(* This function use for BurnerControlEcoFlam
| this version dont have Reset components like Digital output, user have to reset manual at the BurnerControlEcoFlam device
*)
FUNCTION_BLOCK FB_BurnerControlEcoFlam IMPLEMENTS I_BurnerControlEcoFlam

VAR
	piFault	: FB_DigitalInput;
	piFireSussess : FB_DigitalInputExt;
	ifActivePower : I_ActivePower;					//have FB
	ifActivePowerNoFB : I_ActivePowerNoFB;
	eActivePowerType : E_ActivePowerType;
	eState	: E_EcoFlamState;
	bAbort: BOOL;
	bBusy: BOOL;
	bInit: BOOL;
	bReset: BOOL;
	bStop: BOOL;
	bError : BOOL;
	tMeasurement	: TIME := T#200S;
	bIgnition: BOOL;
	bIgnitioned: BOOL;
	tonMeasurementTimer: Ton;
	tBurnSuccess: TIME;
	sName : STRING;
END_VAR

bError := piFault.In; //OR piFireSussess.ErrorTimedout;
piFireSussess();
StateMachine();
tonMeasurementTimer(PT := tMeasurement);
IF piFireSussess.RisingTrigger AND eState = ECOFLAM_IGNITION THEN
	tBurnSuccess	:= 	tonMeasurementTimer.ET;				
END_IF

PROPERTY ActivePowerType : Reference to E_ActivePowerType
GET
ActivePowerType ref= eActivePowerType;
END_GET
END_PROPERTY

{attribute 'monitoring' := 'variable'}
PROPERTY Busy : reference to bool
GET
Busy ref= bBusy;
END_GET
END_PROPERTY

PROPERTY Error : REFERENCE to bool
GET
error REF= bError;
END_GET
END_PROPERTY

{attribute 'monitoring' := 'variable'}
PROPERTY IgnitionSucess : bool
GET
CASE eActivePowerType OF
	ACTIVE_POWER_TYPE_NO_FEEDBACK:
		IgnitionSucess := piFireSussess.In AND ifActivePowerNoFB.PowerOnIsCalled;
		
	ACTIVE_POWER_TYPE_FEEDBACK:
		IgnitionSucess := piFireSussess.In AND ifActivePower.PowerOnIsCalled;
END_CASE
END_GET
END_PROPERTY

PROPERTY Inited : bool
GET
Inited := eState=ECOFLAM_READY_INITIALIZED;
END_GET
END_PROPERTY

PROPERTY IsRefActivePower : bool
GET
IsRefActivePower := ifActivePower<>0 OR ifActivePowerNoFB<>0;
END_GET
END_PROPERTY

PROPERTY IsStop : bool
GET
CASE eActivePowerType OF
	ACTIVE_POWER_TYPE_NO_FEEDBACK:
		isStop := ifActivePowerNoFB.PowerOffIsCalled;
		
	ACTIVE_POWER_TYPE_FEEDBACK:
		isStop := NOT ifActivePower.Powered;
END_CASE
END_GET
END_PROPERTY

METHOD MR_Abort : BOOL
VAR_INPUT
END_VAR
IF eState >= ECOFLAM_INITIALIZING THEN
	bAbort := TRUE;
	bBusy := TRUE;
	MR_Abort := FALSE;
	eState := ECOFLAM_ABORTING;
ELSIF eState = ECOFLAM_UNINITIALIZED THEN
	bAbort := FALSE;
	bBusy := FALSE;
	MR_Abort := TRUE;
END_IF
END_METHOD

METHOD MR_AppendPowerOn : BOOL
VAR_INPUT
	iPowerON	: I_ActivePower;
END_VAR
IF THIS^.ifActivePower <> iPowerON THEN
	THIS^.ifActivePower := iPowerON;
	MR_AppendPowerOn := true;
END_IF
END_METHOD

METHOD MR_AppendPowerOnNoFB : BOOL
VAR_INPUT
	iPowerOnNoFB	: I_ActivePowerNoFB;
END_VAR
IF THIS^.ifActivePowerNoFB <> iPowerOnNoFB THEN
	THIS^.ifActivePowerNoFB := iPowerOnNoFB;
	MR_AppendPowerOnNoFB := true;
END_IF
END_METHOD

METHOD MR_ChooseIfActivePowerType : BOOL
VAR_INPUT
	eChoseActivePowerType : E_ActivePowerType;
END_VAR
eActivePowerType := eChoseActivePowerType;
END_METHOD

METHOD MR_FirstCycle : BOOL
VAR_INPUT
	sName 							: STRING;
	sPiFireSuccessModuleType		: STRING;
	sPiFirePortID					: STRING;
	sPiFaultModuleType				: STRING;
	sPiFaultPortID					: STRING;
	tONBurnerTimeOut				: TIME;
END_VAR
THIS^.sName := sName;
THIS^.piFireSussess.MR_FirstCycleEx(
 	sName			:= CONCAT(sName,':FireSuccess SS'),
	sModuleType 	:= sPiFireSuccessModuleType,
	sPortID			:= sPiFirePortID,
	bEnableTimeout	:= TRUE,
	tDefaultTimeout	:= tONBurnerTimeOut
);
										
THIS^.piFault.MR_FirstCycle(
	sName := CONCAT(sName,':Fault SS'),
	sModuleType := sPiFaultModuleType,
	sPortID := sPiFaultPortID
);
END_METHOD

METHOD MR_Ignition : BOOL
VAR_INPUT
END_VAR
CASE eActivePowerType OF
	ACTIVE_POWER_TYPE_NO_FEEDBACK:
		IF eState = ECOFLAM_READY_INITIALIZED AND NOT ifActivePowerNoFB.PowerOnIsCalled THEN
			bIgnition	:= TRUE;
			MR_Ignition := FALSE;
			bIgnitioned	:= FALSE;
			eState := ECOFLAM_IGNITION;
			bBusy := TRUE;
		ELSIF eState = ECOFLAM_IGNITION_DONE THEN
			bIgnition := FALSE;
			bIgnitioned	:= TRUE;
			MR_Ignition := TRUE;
			bBusy := false	;
		END_IF
		
	ACTIVE_POWER_TYPE_FEEDBACK:
		IF eState = ECOFLAM_READY_INITIALIZED AND NOT ifActivePower.PowerOnIsCalled THEN
			bIgnition	:= TRUE;
			MR_Ignition := FALSE;
			bIgnitioned	:= FALSE;
			eState := ECOFLAM_IGNITION;
			bBusy := TRUE;
		ELSIF eState = ECOFLAM_IGNITION_DONE THEN
			bIgnition := FALSE;
			bIgnitioned	:= TRUE;
			MR_Ignition := TRUE;
			bBusy := false	;
		END_IF
END_CASE
END_METHOD

METHOD  MR_Init : bool // just Acknowledge already append the I_activepower
VAR_INPUT
END_VAR
IF eState = ECOFLAM_UNINITIALIZED THEN
	bInit := TRUE;
	bBusy := TRUE;
	MR_Init := FALSE;
	eState := ECOFLAM_INITIALIZING;
ELSIF eState = ECOFLAM_READY_INITIALIZED THEN
	bInit := FALSE;
	MR_Init := TRUE;
	bBusy := false;
END_IF
END_METHOD

METHOD MR_Reset : BOOL
VAR_INPUT
END_VAR
IF eState >= ECOFLAM_READY_INITIALIZED AND bError THEN
	bBusy := TRUE;
	bReset := TRUE;
	MR_Reset := FALSE;
	eState := ECOFLAM_RESET;
ELSIF eState = ECOFLAM_RESET_DONE THEN
	bBusy := TRUE;
	bReset := FALSE;
	MR_Reset := TRUE;
END_IF
END_METHOD

METHOD MR_Stop : BOOL
VAR_INPUT
END_VAR
CASE eActivePowerType OF
	ACTIVE_POWER_TYPE_NO_FEEDBACK:
		IF eState >= ECOFLAM_INITIALIZING 
			AND eState < ECOFLAM_STOP_DONE 
			AND ifActivePowerNoFB.PowerOnIsCalled  
		THEN
			bStop := true;
			MR_Stop := FALSE;
			bBusy := TRUE;
			eState := ECOFLAM_STOP;
		ELSIF eState = ECOFLAM_STOP_DONE THEN
			bStop := FALSE;
			MR_Stop := TRUE;
			bBusy := false;
		END_IF 
		
	ACTIVE_POWER_TYPE_FEEDBACK:
		IF eState >= ECOFLAM_INITIALIZING 
			AND eState < ECOFLAM_STOP_DONE 
			AND ifActivePower.Powered  
		THEN
			bStop := true;
			MR_Stop := FALSE;
			bBusy := TRUE;
			eState := ECOFLAM_STOP;
		ELSIF eState = ECOFLAM_STOP_DONE THEN
			bStop := FALSE;
			MR_Stop := TRUE;
			bBusy := false;
		END_IF 
END_CASE
END_METHOD

METHOD PROTECTED  MS_Aborting
CASE eActivePowerType OF
	ACTIVE_POWER_TYPE_NO_FEEDBACK:
		ifActivePowerNoFB.MR_PowerOFF();
		piFireSussess.MR_Abort();
		IF NOT piFireSussess.Active THEN
			eState := ECOFLAM_UNINITIALIZED;
		END_IF
		
	ACTIVE_POWER_TYPE_FEEDBACK:
		ifActivePower.MR_PowerOFF();
		piFireSussess.MR_Abort();
		IF NOT ifActivePower.Powered 
			AND NOT ifActivePower.Busy 
			AND NOT piFireSussess.Active
		THEN
			eState := ECOFLAM_UNINITIALIZED;
		END_IF
END_CASE
END_METHOD

METHOD PROTECTED MS_Ignition
VAR_INPUT
END_VAR
CASE eActivePowerType OF
	ACTIVE_POWER_TYPE_NO_FEEDBACK:
		ifActivePowerNoFB.MR_PowerON();
		piFireSussess.MR_StartTracking();
		tonMeasurementTimer.IN := TRUE;
		IF piFireSussess.In  THEN
			eState := ECOFLAM_IGNITION_DONE;
		END_IF
		
	ACTIVE_POWER_TYPE_FEEDBACK:
		ifActivePower.MR_PowerON();
		piFireSussess.MR_StartTracking();
		tonMeasurementTimer.IN := TRUE;
		IF ifActivePower.Powered AND NOT ifActivePower.Busy 
		AND  piFireSussess.In  THEN
			eState := ECOFLAM_IGNITION_DONE;
		END_IF
END_CASE
END_METHOD

METHOD PROTECTED MS_IgnitionDone : BOOL
VAR_INPUT
END_VAR
tonMeasurementTimer.IN := false;
IF NOT bIgnition THEN
	eState :=  ECOFLAM_READY_INITIALIZED;
END_IF
END_METHOD

METHOD PROTECTED MS_Initializing
piFireSussess.MR_Init();
piFireSussess.EnableTimeout := TRUE;

CASE eActivePowerType OF
	ACTIVE_POWER_TYPE_NO_FEEDBACK:
		IF ifActivePowerNoFB <> 0
			AND piFireSussess.Active
		THEN
			eState := ECOFLAM_READY_INITIALIZED;
		END_IF
		
	ACTIVE_POWER_TYPE_FEEDBACK:
		IF ifActivePower <> 0
			AND piFireSussess.Active
		THEN
			eState := ECOFLAM_READY_INITIALIZED;
		END_IF
END_CASE
END_METHOD

METHOD PROTECTED MS_ReadyInitialized
VAR_INPUT
END_VAR
bBusy := false;
END_METHOD

(*
this version just reset piFireSussess, User have to reset manually at the device
*)
METHOD PROTECTED MS_Reset : BOOL
piFireSussess.MR_Reset();
bInit 		:= FALSE;
bAbort		:= FALSE;
bIgnition 	:= FALSE;
bStop 		:= FALSE;
IF NOT piFireSussess.ErrorTimedout THEN
	eState := ECOFLAM_RESET_DONE;
END_IF
END_METHOD

(* don't not edit*)
METHOD PROTECTED MS_ResetDone
VAR_INPUT
END_VAR
eState := ECOFLAM_READY_INITIALIZED;
END_METHOD

METHOD protected MS_Stop 
VAR_INPUT
END_VAR
CASE eActivePowerType OF
	ACTIVE_POWER_TYPE_NO_FEEDBACK:
		ifActivePowerNoFB.MR_PowerOFF();
		eState := ECOFLAM_STOP_DONE;
		
	ACTIVE_POWER_TYPE_FEEDBACK:
		ifActivePower.MR_PowerOFF();
		IF NOT ifActivePower.Powered AND not ifActivePower.Busy THEN
			eState := ECOFLAM_STOP_DONE;
		END_IF
END_CASE
END_METHOD

METHOD protected Ms_StopDone
VAR_INPUT
END_VAR
IF NOT bStop THEN
	eState := ECOFLAM_READY_INITIALIZED;
END_IF
END_METHOD

METHOD PROTECTED MS_Uninitialized
bBusy := FALSE;

piFireSussess.EnableForce := FALSE;
piFireSussess.EnableTimeout := FALSE;

bInit 		:= FALSE;
bReset		:= FALSE;
bAbort		:= FALSE;
END_METHOD

PROPERTY Name : string
GET
Name := sName;
END_GET
SET
sName := Name;
END_SET
END_PROPERTY

PROPERTY Ref_IfActivePower : REFERENCE TO I_ActivePower
GET
Ref_IfActivePower ref= ifActivePower;
END_GET
END_PROPERTY

PROPERTY Ref_IfActivePowerNoFB : REFERENCE TO I_ActivePowerNoFB
GET
Ref_IfActivePowerNoFB ref= ifActivePowerNoFB;
END_GET
END_PROPERTY

PROPERTY Ref_piFault : reference to  FB_DigitalInput
GET
ref_piFault ref= piFault;
END_GET
END_PROPERTY

PROPERTY Ref_piIgnitionSucess : reference to  FB_DigitalInput
GET
ref_piIgnitionSucess ref= piFireSussess;
END_GET
END_PROPERTY

PROPERTY State : E_EcoFlamState
GET
State := eState;
END_GET
END_PROPERTY

METHOD PROTECTED StateMachine
CASE eState OF
	ECOFLAM_UNINITIALIZED :
		MS_Uninitialized();
		
	ECOFLAM_INITIALIZING	:
		MS_Initializing();
		
	ECOFLAM_READY_INITIALIZED :
		MS_ReadyInitialized();
		
	ECOFLAM_IGNITION	:
		MS_Ignition();
		
	ECOFLAM_IGNITION_DONE	:
		MS_IgnitionDone();
		
	ECOFLAM_STOP		:
		MS_Stop();
		
	ECOFLAM_STOP_DONE	:
		Ms_StopDone();
		
	ECOFLAM_RESET:
		MS_Reset();
		
	ECOFLAM_RESET_DONE:
		MS_ResetDone();
		
	ECOFLAM_ABORTING :
		MS_Aborting();
	
END_CASE
END_METHOD

END_FUNCTION_BLOCK

(* stored: Version 1.1.0.1, ProductVersion 3.1.4024.12
   POU FB_BurnerControlEcoFlam: Id {88a4ffff-4393-4d36-8255-c49816de1886}, SpecialFunc None
   Folder Internal: Id {f26a0759-c8bf-493c-864a-44e8b610bce1}
   Folder Properties: Id {a2727e65-94e4-494e-9e3d-2cd8c9e1e5a1}
   Folder Request: Id {81afbd00-65cb-4926-838a-d602e3a1ed61}
   Property ActivePowerType: Id {d9badd35-a76a-476f-bed8-2ef6932be687}
   Get Get: Id {91a63427-0abe-49a7-a4c8-600b2d1183b5}
   Property Busy: Id {fef0549e-1f99-4a56-ac1c-5f5b496a688e}
   Get Get: Id {5f87b202-0648-4783-bd0c-e6dd9d5246e1}
   Property Error: Id {1292a722-8fad-4cb4-8af9-bc6a89fba151}
   Get Get: Id {8d356e25-bf04-40e5-8279-0e1f0e525a86}
   Property IgnitionSucess: Id {34b96f87-b0ab-4802-bed2-5c8e059abd23}
   Get Get: Id {3a7d24d9-82de-4909-8b4b-de5975f43f67}
   Property Inited: Id {77fbaf7a-0a5e-49c6-8cfa-cac730d2a1e3}
   Get Get: Id {e9c44e9b-d3d7-4315-bb12-fadae2e3dd49}
   Property IsRefActivePower: Id {a6ad5d9a-0822-4162-adc5-bcaef2e2d72c}
   Get Get: Id {92ae821a-21ee-4325-ab66-71548c130800}
   Property IsStop: Id {f5f1fb6b-1e47-4c5e-b372-bbc55886a0c6}
   Get Get: Id {0981c464-f7c3-4ed6-9bbb-d69c78ebaff5}
   Method MR_Abort: Id {1f1cc6f1-0a14-4d5f-b2ff-67ddc8a3b880}
   Method MR_AppendPowerOn: Id {0ed5ced2-0827-4e45-b64a-410e2eb14889}
   Method MR_AppendPowerOnNoFB: Id {854162b0-71e4-48c5-bf1a-0aa214361348}
   Method MR_ChooseIfActivePowerType: Id {a1c802e6-0c05-4e5e-8272-911357a7f46d}
   Method MR_FirstCycle: Id {675c34c3-dfa8-4d52-b1c0-aa64a4ad7181}
   Method MR_Ignition: Id {49a25cbf-788a-4dc3-a129-f90e295a4b26}
   Method MR_Init: Id {b73be3d0-0d4d-418a-928d-8354a1d399c2}
   Method MR_Reset: Id {9dbbb7c6-b46a-4998-9cc0-fb272acc39ab}
   Method MR_Stop: Id {e2d68bec-bb32-4b9d-b877-becb5ffec602}
   Method MS_Aborting: Id {a07ebe05-4cbc-43cb-8e7f-81ee4594d53b}
   Method MS_Ignition: Id {91633012-c724-40b7-94f9-37b2aa1a449f}
   Method MS_IgnitionDone: Id {fcded8cd-1c5d-4265-8ef9-ee72d739d61a}
   Method MS_Initializing: Id {c1a3196a-3075-45ae-936b-345730e3d6c3}
   Method MS_ReadyInitialized: Id {e01c8096-984a-42e6-80c7-cd403967703e}
   Method MS_Reset: Id {ce905759-3b28-40ed-a33c-aa295b63c877}
   Method MS_ResetDone: Id {f943014d-068b-4845-bb11-9f41ba5be81e}
   Method MS_Stop: Id {0427a35e-52cf-4579-b5b6-38d6e9db201d}
   Method Ms_StopDone: Id {7edb9d39-a958-4e60-a247-b79d4f8bd4e2}
   Method MS_Uninitialized: Id {cfae14a1-1329-4d0a-b581-62d0426a1451}
   Property Name: Id {e896ae50-e3d1-4588-b4af-4158a7bc28a6}
   Get Get: Id {59f9f528-157a-4d80-9ac5-1503c993dcca}
   Set Set: Id {ab4d986b-3ca0-4d87-8bf0-c0f77b5e2bc3}
   Property Ref_IfActivePower: Id {a332cb4a-3c3c-4e12-942d-2f2c9a5f5fe6}
   Get Get: Id {db58f3bc-0ca6-4727-b5d0-cfda39ecc22d}
   Property Ref_IfActivePowerNoFB: Id {4e7021cf-5bd8-4dc9-9752-e0985fa2850d}
   Get Get: Id {f7a8eed8-d0fa-4a64-b764-348ec7937ff5}
   Property Ref_piFault: Id {7257d8a2-cf6d-41d9-b51a-05975eb8a988}
   Get Get: Id {bdef0ba5-b065-4461-84d0-2f6ce92c5c44}
   Property Ref_piIgnitionSucess: Id {f2931f18-cca9-4eb3-bf1b-a96e57bdf70d}
   Get Get: Id {6264c58a-ea7e-4735-9bd0-b2e41557bb44}
   Property State: Id {7ca2aba7-6ae1-4c02-9a13-353f42db7c21}
   Get Get: Id {c815f0b1-e767-4975-80bb-0430a1e3c989}
   Method StateMachine: Id {f939ecf1-c196-4392-9843-2153cb9c76fe} *)
